PROGRAM Tcp_ip
VAR
	bConnect: BOOL;
	bRecieve: BOOL;
	FB_create: FB_SocketUdpCreate;
	FB_Recieve: FB_SocketUdpReceiveFrom;
	FB_close: FB_SocketClose;
	data : ARRAY[0..500] OF BYTE;
END_VAR

FB_create(
	sSrvNetId:= , 							//Lokaal netwerk (mag leeg blijven)
	sLocalHost:= '127.0.0.1', 			//Eigen ip van de PC en ingesteld in de gateway
	nLocalPort:= 8080,						//Ingesteld op de gateway
	bExecute:= bConnect,					//Trigger voor functieblok
	tTimeout:= T#1S);
	

FB_Recieve(
	sSrvNetId:= , 									//Lokaal netwerk (mag leeg blijven)
	hSocket:= FB_create.hSocket,					 
	cbLen:= SIZEOF(data), 							//Kijkt naar de lengte van het bericht
	pDest:= ADR(data), 								//Plaat waar de het bericht wordt opgeslaan
	bExecute:= NOT FB_recieve.bBusy AND bRecieve, 	//Trigger voor functieblok
	tTimeout:= T#1S);
	
FB_close(
	sSrvNetId:= , 							//Lokaal netwerk (mag leeg blijven)
	hSocket:= FB_create.hSocket, 			
	bExecute:= NOT bConnect, 				//Sluiten van de connectie 
	tTimeout:= T#1S);
	
IF FB_Recieve.nRecBytes > 0 THEN 										//Dit gebuert op het moment dat er data binnenkomt
	memcpy(ADR(GVL.sDatastring),ADR(data),FB_Recieve.nRecBytes);			//Het bericht zal worden opgeslaan in Datastring
	memcpy(ADR(GVL.sDatastring) + FB_Recieve.nRecBytes,ADR(GVL.NullByte),1);	//Nullbyte word gedetecteerd stoppen met bericht plaatsen
	Decoder();

END_IF

END_PROGRAM

(* stored: Version 1.1.0.1, ProductVersion 3.1.4024.0
   POU Tcp_ip: Id {93165edd-5589-407a-ae5c-9a5ae0ff5f10}, SpecialFunc None *)
